INTERFACE I_Module

METHOD PUBLIC GetLastErrorMessage : T_MAXSTRING
VAR_INPUT
END_VAR
END_METHOD

PROPERTY PUBLIC HasError : BOOL
GET
END_GET
END_PROPERTY

PROPERTY PUBLIC Name : T_MAXSTRING
GET
END_GET
END_PROPERTY

END_INTERFACE

(* stored: Version 1.1.0.1, ProductVersion 3.1.4024.12
   Itf I_Module: Id {42a26287-dd54-4ea0-b34f-f9f119ef00c5}
   Method GetLastErrorMessage: Id {a039a7cd-6211-401b-9e8c-b5534efdf5c4}
   Property HasError: Id {a2104551-6386-44fe-9548-fe24f493936b}
   Get Get: Id {5d42d25e-de91-4b70-b7e8-797214bc4924}
   Property Name: Id {4b8b783f-f896-45aa-a663-9468161d78f3}
   Get Get: Id {68dc8ed6-60c9-4d7a-8486-57df30d5fc62} *)
